{attribute 'Tc2GvlVarNames'}
VAR_GLOBAL
	
	Cellule_mesure_barre					:BOOL;

END_VAR

(* stored: Version 1.1.0.1, ProductVersion 3.1.4024.15
   GVL IO_BE: Id {bb6b04a5-ef2c-4824-a73e-0c9dd5e4fe12} *)
